FUNCTION_BLOCK PKP_2200_LI_4_DI (* Service Interface Function Block Type *)
  (* Standard: SAE J1939; Function: Combo Block: 8 Inputs/8 Outputs (includes all input/output types); Type: DP-34044-1-000; Description: this maps to IX/QX *)
  (* Version 1.0, 2018-12-05, Jose Cabral *)
  (* Version 1.1, 2022-08-04, Franz Höpfinger, HR Agrartechnik GmbH *)
  (* Version 1.2, 2023-01-05, Franz Höpfinger, HR Agrartechnik GmbH *)
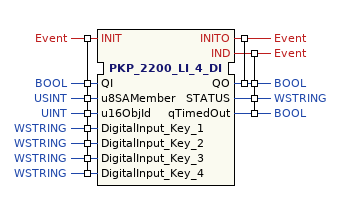
  EVENT_INPUT
    INIT WITH QI, u8SAMember, u16ObjId, DigitalInput_Key_1, DigitalInput_Key_2, DigitalInput_Key_3, DigitalInput_Key_4; (* Service Initialization *)
  END_EVENT
  EVENT_OUTPUT
    INITO WITH QO; (* Initialization Confirm *)
    IND WITH QO, STATUS, qTimedOut; (* Indication from Resource *)
  END_EVENT
  VAR_INPUT
    QI : BOOL; (* Event Input Qualifier *)
    u8SAMember : USINT := 224; (* Node SA Default 21h *)
    u16ObjId : UINT := 65535; (* Dummy ! set to 65535 if in Doubt. 0 deactivates FB. *)
    DigitalInput_Key_1 : WSTRING := "DigitalInput_Key_1";
    DigitalInput_Key_2 : WSTRING := "DigitalInput_Key_2";
    DigitalInput_Key_3 : WSTRING := "DigitalInput_Key_3";
    DigitalInput_Key_4 : WSTRING := "DigitalInput_Key_4";
  END_VAR
  VAR_OUTPUT
    QO : BOOL; (* Event Output Qualifier *)
    STATUS : WSTRING; (* Service Status *)
    qTimedOut : BOOL;
  END_VAR
END_FUNCTION_BLOCK
